{attribute 'Tc2GvlVarNames'}
VAR_GLOBAL CONSTANT
	(* Pumpe_Zustand_Status *)
	E_PU_Zustand_Status_Idle_Sperre			: SINT := 0;
	E_PU_Zustand_Status_Betriebsbereit		: SINT := 1;
	E_PU_Zustand_Status_Nachl				: SINT := 2;
	E_PU_Zustand_Status_Vorl				: SINT := 3;
	E_PU_Zustand_Status_Betrieb				: SINT := 4;
	E_PU_Zustand_Status_Betrieb_Sperre		: SINT := 5;
	E_PU_Zustand_Status_Stoerung			: SINT := 99;

	(* Pumpe_Zustand_Regelung_Modus *)
	E_PU_Regelung_Modus_P					: SINT := 0;
	E_PU_Regelung_Modus_dT					: SINT := 1;
	E_PU_Regelung_Modus_dT_invert			: SINT := 2;
	E_PU_Regelung_Modus_T_int				: SINT := 3;
	E_PU_Regelung_Modus_T_ext				: SINT := 4;
	E_PU_Regelung_Modus_dp_auto				: SINT := 5;
END_VAR

(* stored: Version 1.1.0.1, ProductVersion 3.1.4024.9
   GVL Con_PU: Id {a122b55e-adf8-466e-ae95-3491c242219e} *)
